PROGRAM main
  VAR
    sensor AT %IX0.0 : BOOL;
    conveyor_run AT %QX0.0 : BOOL;
    object_arrived AT %QX0.1 : BOOL;
    pick_done AT %QX0.2 : BOOL;
  END_VAR

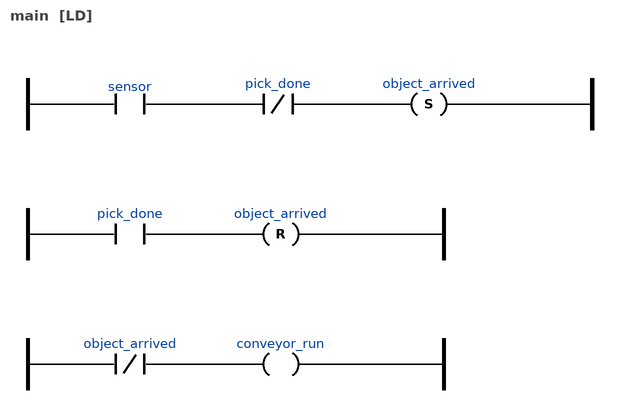
(* LD diagram, written out as Structured Text *)
IF sensor AND NOT pick_done THEN object_arrived := TRUE; END_IF;
IF pick_done THEN object_arrived := FALSE; END_IF;
conveyor_run := NOT object_arrived;
END_PROGRAM
